(* IEC 61131-3 sources: Industry-PLC-LLM/data/PLCBEAD_repo/PLCBEAD_PLCEmbed-main/PLC-BEAD/Source/GEB/TOD_TO_TIME, 1 file *)

(* ---- TOD_TO_TIME.ST ---- *)
FUNCTION TOD_TO_TIME2:TIME
	VAR_INPUT
		IN :	UDINT;
	END_VAR

	TOD_TO_TIME2 := DWORD_TO_TIME(UDINT_TO_DWORD(IN));
END_FUNCTION

PROGRAM program0
  VAR
	IN :	UDINT;
    CEIL5_OUT : TIME;
  END_VAR

  CEIL5_OUT := TOD_TO_TIME2(IN);
END_PROGRAM
